Staubli VAL3: crc16.pgx

program crc16(num n, num& rh, num& rl, num& buf[])
  local num Poly
  local num i
  local num j
  local num crc
  local num carry
begin

//*******************************************************************************
//*   ______
//*  / _____) /|
//* | |      / /
//* | | /\  / /
//* | | \ \/ /  _      Copyright (c) KEOLABS, 2016
//* | |  \__/  | |        http://www.keolabs.com
//* | |________| |
//*  \__________/
//*
//********************************************************************************
//*@file          : crc16
//*@author        : Yves Ragot
//*@version       : $Id: crc16.pgx 1561 2017-01-06 10:24:51Z yves $
//*@brief         : CRC16 computing of a PC frame
//*
//*******************************************************************************/

  //#define Poly 0xA001
  Poly = 40961

  crc = 65535

  for i = 0 to (n - 1)

      crc = bXor(crc, bAnd(buf[i], 255))

      for j = 0 to 7

          carry = bAnd(crc, 1)
          crc = roundDown(crc / 2)

          if ( carry == 1 )
              crc = bXor(crc, Poly)
          endIf

      endFor

  endFor

  rh = bAnd(crc, 255)
  rl = roundDown(crc / 256)

end
